TYPE OrderTable_DUT :
STRUCT
	OrderNo:  INT;
	StepNo:  INT;
	PlaceTime:  String[20];
	Device:  String;
	Sequence:  UInt;
	Status:  String[12];
	CompleteTime:  String[20];
	ErrorID:  UInt;
	OPC_Control:  WMS_OPC_UA_DUT;
END_STRUCT
END_TYPE

(* stored: Version 1.1.0.1
   DUT OrderTable_DUT: Id {151c6b8a-b953-4881-adb3-0874a151ea14} *)
